{region '#Template'}                                                                                                                                                                                                                                                {region '#Template'}
	{attribute 'Version' := '5.0.0.0'}
	{attribute 'Tags' := '"LCID": "1031", "Text": "Gewerk, Gebäudeautomation"'}
	{attribute 'Tags' := '"LCID": "1033", "Text": "Trade, Building automation"'}
	{attribute 'Using' := '"Type": "Template", "URI": "Site"'}
	{attribute 'Description' := '"LCID": "1031", "Text": "Aufruf der Anlagen des Gewerks Gebäudeautomation"'}
	{attribute 'Description' := '"LCID": "1033", "Text": "Calling the plants of the trade building automation"'}
{endregion}	 
	 
FUNCTION_BLOCK FB_BA_BuildingAutomationServer EXTENDS FB_BA_View
VAR_INPUT CONSTANT
	AdsComServerBasic		: FB_BA_AdsComServer_Basic;	
	Weatherstation01		: FB_BA_WeatherStation_Thies;	
	WeatherData 			: FB_BA_WeatherData;	
END_VAR

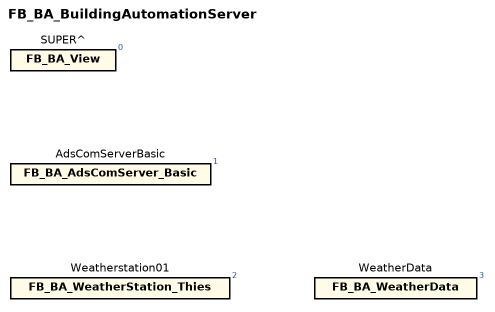
SUPER^(); // FB_BA_View
AdsComServerBasic(); // FB_BA_AdsComServer_Basic
Weatherstation01(); // FB_BA_WeatherStation_Thies
WeatherData(); // FB_BA_WeatherData

METHOD FB_init : BOOL
VAR_INPUT
	bInitRetains : BOOL; // if TRUE, the retain variables are initialized (warm start / cold start)
	bInCopyCode : BOOL;  // if TRUE, the instance afterwards gets moved into the copy code (online change)
END_VAR
Weatherstation01.iParent		:= THIS^;
Weatherstation01.iLabel			:= LblPlt_Weather_station;
Weatherstation01.sObjectName	:= '{Idx=01}';
Weatherstation01.sDescription	:= '{Idx=01}';
Weatherstation01.eDPADMode		:= E_BA_DPADMode.eInclude;

WeatherData.iParent			    := THIS^;
WeatherData.iLabel			    := LblPlt_Weather_data;
WeatherData.sObjectName		    := '{Idx=01}';
WeatherData.eDPADMode		    := E_BA_DPADMode.eInclude;
END_METHOD

END_FUNCTION_BLOCK

(* stored: Version 1.1.0.1, ProductVersion 3.1.4024.12
   POU FB_BA_BuildingAutomationServer: Id {32cf740d-c924-45a7-97a9-050f005fc905}, SpecialFunc None
   Method FB_init: Id {8433a42f-4c6d-43a6-9ce9-8f04da1c59e6} *)
